// TIA Portal V20 export
DATA_BLOCK "HmiInterface"   // DB98
// stored: Access Published, MemoryReserve 100, Namespace Unit1.Em7
   VAR
      em : "LAF_typeEmInterface";
      emHomedCheck : "Unit1.Em7.typeEmHomedCheck";
      cm : "Unit1.Em7.typeCmInterface";
      conveyor : "LER_typeSequenceInterface";
      ngKicker : "LER_typeSequenceInterface";
      passKicker : "LER_typeSequenceInterface";
      qrReaderSTK1 : "LER_typeSequenceInterface";
      qrReaderSTK2 : "LER_typeSequenceInterface";
      InterfaceSTK1 : "LER_typeSequenceInterface";
      InterfaceSTK2 : "LER_typeSequenceInterface";
   END_VAR
   VAR RETAIN
      cmNgKickerAxisZ : "LBC_typeAxisControlInterface";
      cmPassKickerAxisZ : "LBC_typeAxisControlInterface";
      cmCutConveyorAxisB : "LBC_typeAxisControlInterface";
      cmNgConveyorAxisB : "LBC_typeAxisControlInterface";
      cmStack1ConveyorAxisB : "LBC_typeAxisControlInterface";
      cmStack2ConveyorAxisB : "LBC_typeAxisControlInterface";
      cmConveyorVirtualAxisB : "LBC_typeAxisControlInterface";
      cmCutConveyorRingBlow : "LBC_typeSinaSpeedInterface";
      cmNgConveyorRingBlow : "LBC_typeSinaSpeedInterface";
      cmStack2ConveyorRingBlow : "LBC_typeSinaSpeedInterface";
      cmNgBoxLockCylinderUpDown : "LBC_typeTwoWayActuatorInterface";
      cmNgBoxDetectSensor : "LBC_typeDigitalSignalInterface";
      cmNgBoxFullSensor : "LBC_typeDigitalSignalInterface";
      cmNgKickerDetectSensor : "LBC_typeDigitalSignalInterface";
      cmPassKickerDetectSensor : "LBC_typeDigitalSignalInterface";
      cmStack1ConveyorElectrodeDetectSensor : "LBC_typeDigitalSignalInterface";
      cmStack2ConveyorElectrodeDetectSensor : "LBC_typeDigitalSignalInterface";
      cmStack1QrReader : "LER_typeSRX300Interface";
      cmStack2QrReader : "LER_typeSRX300Interface";
      cmNgKickerAxisZ_TorqueCal : "LER_typeServoTorqueCalInterface";
      cmPassKickerAxisZ_TorqueCal : "LER_typeServoTorqueCalInterface";
      cmCutConveyorAxisB_TorqueCal : "LER_typeServoTorqueCalInterface";
      cmNgConveyorAxisB_TorqueCal : "LER_typeServoTorqueCalInterface";
      cmStack1ConveyorAxisB_TorqueCal : "LER_typeServoTorqueCalInterface";
      cmStack2ConveyorAxisB_TorqueCal : "LER_typeServoTorqueCalInterface";
      ngKickerSensorNotDetectedCount : "LER_typeAlarmCounterInterface";
      passKickerSensorNotDetectedCount : "LER_typeAlarmCounterInterface";
      stack1ConveyorElectrodeSensorNotDetectedCount : "LER_typeAlarmCounterInterface";
      stack2ConveyorElectrodeSensorNotDetectedCount : "LER_typeAlarmCounterInterface";
      visionConsecutiveNgOutCount : "LER_typeAlarmCounterInterface";
      cmStack1QrHistory : "LER_typeQrHistory";
      cmStack2QrHistory : "LER_typeQrHistory";
      RingBlow_SleepModeRunPct : Real;
   END_VAR
   VAR
      UserRecoveryPassOkButton : Bool;
   END_VAR
BEGIN
   cmNgKickerAxisZ.commandConfiguration.posAbsolute.velocity := 150.0;
   cmNgKickerAxisZ.commandConfiguration.posAbsolute.acceleration := -1.0;
   cmPassKickerAxisZ.commandConfiguration.posAbsolute.velocity := 150.0;
END_DATA_BLOCK
